VAR_GLOBAL CONSTANT
	cusiMinAddedChilds: USINT := 1;
	cMAX_JAM_SENSORS: USINT := 3;
END_VAR

(* stored: Version 1.1.0.1, ProductVersion 3.1.0.23
   GVL Const_MER: Id {a8b687c4-08ff-4f13-97ef-63a0034a56ce} *)
